# EPICS substitutions: apps/db/userHost.substitutions
# Example substitutions file

file "db/dbExample1.db" {
    { user = "levonHost" }
}

file db/dbExample2.db {
    pattern { user, no, scan }
        { "levonHost", 1, "1 second" }
        { "levonHost", 2, "2 second" }
        { "levonHost", 3, "5 second" }
}
